// TIA Portal V19 export
ORGANIZATION_BLOCK "Startup"   // OB2005, LAD, Startup
TITLE = "Complete Restart"
// stored: AutoNumber false, Namespace Unit.Em0, SetENOAutomatically false
   VAR_INPUT
      LostRetentive : Bool;   // True if retentive data are lost
      LostRTC : Bool;   // True if date and time are lost
   END_VAR
BEGIN

REGION Network 1 (SCL): Build the Absolut Reference Designator
   // Set the Absoult Reference Designator in the Config DB
   IF LEN(IN := "Unit.Em0.Config".em.referenceDesignator.parent) <> 0 THEN
       "Unit.Em0.Config".em.referenceDesignator.combined := CONCAT_WSTRING(IN1 := "Unit.Em0.Config".em.referenceDesignator.parent, IN2 := WSTRING#'.', IN3 := "Unit.Em0.Config".em.referenceDesignator.relative);
   ELSE
       "Unit.Em0.Config".em.referenceDesignator.combined := "Unit.Em0.Config".em.referenceDesignator.relative;
   END_IF;
END_REGION
END_ORGANIZATION_BLOCK
